FUNCTION F_Log3 
VAR_INPUT
	eLogLevel		: E_LogLevel;
	sMessage		: T_MaxString;
	stArg1			: T_Arg;
	stArg2			: T_Arg;
	stArg3			: T_Arg;
END_VAR

F_LogL3(eLogLevel, Const.sGlobalLogger, sMessage, stArg1, stArg2, stArg3);

END_FUNCTION

(* stored: Version 1.1.0.1, ProductVersion 3.1.4024.0
   POU F_Log3: Id {0aaacd3b-494c-4cb5-ab64-7abdca7ffb13}, SpecialFunc None *)
